(* IEC 61131-3 sources: programs/VI-54/VI-54_20171205/VI-54_20171205/Stations/Screen/LseClass170718/Class/CheckOnlineStatus, 1 file *)

(* ---- CheckOnlineStatus.st ---- *)
(*!
<Class
	Name               = "CheckOnlineStatus"
	Revision           = "1.0"
	RealtimeTask       = "false"
	CyclicTask         = "true"
	DefCyclictime      = "50 ms"
	BackgroundTask     = "false"
	Sigmatek           = "false"
	OSInterface        = "false"
	HighPriority       = "false"
	Automatic          = "false"
	UpdateMode         = "Prescan"
	SharedCommandTable = "true"
	Objectsize         = "(600,180)"
	Comment            = "class for checking/alarming the online status">
	<Channels>
		<Server Name="AlarmState" Visualized="true" Initialize="false" WriteProtected="false" Retentive="false" Comment="actual status of the communication alarm"/>
		<Server Name="Locked" Visualized="false" Initialize="false" WriteProtected="true" Retentive="false" Comment="0 ... communication never was online&#13;&#10;1 ... communication was online -&gt; alarming enabled"/>
		<Client Name="AlarmCommunication" Required="true" Internal="true"/>
		<Client Name="AlarmNo" Required="true" Internal="false" Comment="alarm number for PLC offline alarm (input)"/>
		<Client Name="toTCPComm" Required="true" Internal="false" Comment="Object channel to TCPCommunication."/>
	</Channels>
	<RevDoku>
		<Owner Company="Sigmatek"/>
		<Dokumentation Revision="1.0" Date="2015-06-24" Company="Sigmatek" Description="Creation."/>
	</RevDoku>
	<Network Name="CheckOnlineStatus">
		<!-- List of Components in this network -->
		<Components>
			<Object
				Name       = "AlarmCommunication"
				Class      = "_AlarmX0Para"
				Position   = "(210,240)"
				Visualized = "true">
				<Channels>
					<Server Name="ClassSvr"/>
					<Client Name="Acknow"/>
					<Client Name="Config" Value="0"/>
					<Client Name="Group"/>
				</Channels>
			</Object>
		</Components>
		<Comments>
		</Comments>
		<!-- List of Connections in this network -->
		<Connections>
			<Connection Source="AlarmCommunication.Config" Destination="this.AlarmNo" Vertices="(210,330),(38,270),"/>
			<Connection Source="this.AlarmState" Destination="AlarmCommunication.ClassSvr" Vertices="(938,270),(766,330),"/>
			<Connection Source="this.AlarmCommunication" Destination="AlarmCommunication.ClassSvr"/>
		</Connections>
		<!-- Headerfiles -->
		<Options>
		</Options>
	</Network>
</Class>
*)
CheckOnlineStatus : CLASS
  //Servers:
	Locked 	: SvrChCmd_DINT;
	AlarmState 	: SvrCh_DINT;
  //Clients:
	toTCPComm 	: CltChCmd_TCPCommunication;
	AlarmNo 	: CltCh_DINT;
	AlarmCommunication 	: CltChCmd__AlarmX0Para;
  //Variables:
  //Functions:

	FUNCTION VIRTUAL GLOBAL CyWork
		VAR_INPUT
			EAX 	: UDINT;
		END_VAR
		VAR_OUTPUT
			state (EAX) 	: UDINT;
		END_VAR;

	FUNCTION VIRTUAL GLOBAL AlarmState::Read
		VAR_OUTPUT
			output (EAX) 	: DINT;
		END_VAR;

	FUNCTION VIRTUAL GLOBAL AlarmState::Write
		VAR_INPUT
			input (EAX) 	: DINT;
		END_VAR
		VAR_OUTPUT
			result (EAX) 	: DINT;
		END_VAR;
  //Tables:
	FUNCTION @STD
		VAR_OUTPUT
			ret_code	: CONFSTATES;
		END_VAR;
	FUNCTION GLOBAL TAB @CT_;
END_CLASS;

#pragma using _AlarmX0Para
#pragma usingLtd TCPCommunication

FUNCTION VIRTUAL GLOBAL CheckOnlineStatus::CyWork
	VAR_INPUT
		EAX 	: UDINT;
	END_VAR
	VAR_OUTPUT
		state (EAX) 	: UDINT;
	END_VAR

  // Warten bis Kommunikation Online ist
  //---------------------------------------------------
  if Locked = 0 then

    if toTCPComm.Online then
      Locked := 1;
    end_if;

  // Kommunikation ist Online
  //---------------------------------------------------
  else

    if toTCPComm.Online then

      if toTCPComm.TransferRateReceive <> 0 then
        // online
        if AlarmCommunication.ClassSvr.Read() <> 0 then
          AlarmCommunication.ClassSvr.Write(input:=0);
        end_if;

      else
        // offline
        if AlarmCommunication.ClassSvr.Read() <> 1 then
          AlarmCommunication.ClassSvr.Write(input:=1);
        end_if;
      end_if;

    else

      // offline
      if AlarmCommunication.ClassSvr.Read() <> 1 then
        AlarmCommunication.ClassSvr.Write(input:=1);
      end_if;

    end_if;

  end_if;

	state := READY;

END_FUNCTION

FUNCTION VIRTUAL GLOBAL CheckOnlineStatus::AlarmState::Read
	VAR_OUTPUT
		output (EAX) 	: DINT;
	END_VAR

	AlarmState := AlarmCommunication.ClassSvr.Read();
	output := AlarmState;

END_FUNCTION

FUNCTION VIRTUAL GLOBAL CheckOnlineStatus::AlarmState::Write
	VAR_INPUT
		input (EAX) 	: DINT;
	END_VAR
	VAR_OUTPUT
		result (EAX) 	: DINT;
	END_VAR

	AlarmState := input;
	result := (AlarmCommunication.ClassSvr.Write(AlarmState))$DINT;

END_FUNCTION
